(* IEC 61131-3 sources: eCockpitGit/test_project/src/%PLC%PLCTest2/%PLOG%Plc Logic/%APP%APP1_Test/%F%NormalFolder/%ITF%ITF_1, 1 file *)

(* ---- %METH%METHski.st ---- *)
METHOD METHski
VAR_INPUT
	test:INT;
END_VAR

(*%!%__DELIMITER__%!%*)
